// TIA Portal project "Alojado_FillingTank_FactoryIO" (V16)

(* hardware
DEVICE "S7-1200 station_1"  S7-1200 Station
   slot 0: "Rack_0"  S7-1200 Rack  Rack  V1.0
   slot 1: "PLC_1"  CPU 1215C DC/DC/DC  6ES7 215-1AG40-0XB0  V4.4
*)

// ===== PLC "PLC_1"  CPU 1215C DC/DC/DC =====

VAR_GLOBAL   // PLC tag table "Default tag table"
   "Tag_5" AT %M0.0 : Bool;
   "Tag_8" AT %M0.1 : Bool;
   "Tag_9" AT %MD10 : DInt;
   "Tag_10" AT %MD14 : DInt;
   "Tag_11" AT %MD18 : DInt;
   "Tag_1" AT %M0.2 : Bool;
   "Tag_12" AT %M0.3 : Bool;
   "Tag_13" AT %MD22 : Time;
   "Tag_14" AT %MD26 : DInt;
   "Tag_15" AT %MD30 : DInt;
END_VAR

VAR_GLOBAL   // PLC tag table "Tag table from XML_3"
   "Fill PB" AT %I10.0 : Bool;
   "Discharge PB" AT %I10.1 : Bool;
   "FACTORY I/O (Running)" AT %I10.2 : Bool;
   "Fill valve" AT %Q0.0 : Bool;
   "Filling Light" AT %Q0.1 : Bool;
   "Discharge valve" AT %Q0.2 : Bool;
   "Discharging Light" AT %Q0.3 : Bool;
   "Timer" AT %QD30 : DInt;
END_VAR

// folder: System blocks/Program resources

DATA_BLOCK "IEC_Timer_0_DB"   // DB1
{ S7_Optimized_Access := 'TRUE' }
AUTHOR : Simatic
FAMILY : IEC
NAME : IEC_TMR
VERSION : 1.0
// stored: InstanceOfName IEC_TIMER
"IEC_TIMER"
BEGIN
END_DATA_BLOCK

DATA_BLOCK "IEC_Timer_0_DB_1"   // DB2
{ S7_Optimized_Access := 'TRUE' }
AUTHOR : Simatic
FAMILY : IEC
NAME : IEC_TMR
VERSION : 1.0
// stored: InstanceOfName IEC_TIMER
"IEC_TIMER"
BEGIN
END_DATA_BLOCK

// folder: (top level)

FUNCTION "MHJ-PLC-Lab-Function-S71200" : Void   // FC9000, SCL
{ S7_Optimized_Access := 'TRUE' }
VERSION : 0.1
   VAR_TEMP
      rdTimeReturn : Int;
      outputTime : DTL;
      SyncVal : Byte;
      forVal : Int;
      forVal_2 : Int;
      Value : Byte;
   END_VAR
   VAR CONSTANT
      CompVal : Byte := 16#34;
      Value_01 : Byte := 16#11;
      Value_01_DW : DWord := 16#A165_D992;
      Value_02_DW : DWord := 16#58BE_4401;
   END_VAR
BEGIN

   #Value:=PEEK(area := 16#82,
        dbNumber := 0,
        byteOffset := 511);
   #Value := #Value + 1;

   POKE(area := 16#82,
        dbNumber := 0,
        byteOffset := 511,
        value := #Value);

   POKE(area:=16#81,
        dbNumber:=0,
        byteOffset:=1016,
        value:=#Value_01_DW);
   POKE(area := 16#81,
        dbNumber := 0,
        byteOffset := 1020,
        value := #Value_02_DW);

   POKE(area := 16#81,
        dbNumber := 0,
        byteOffset := 511,
        value := B#16#00);

   FOR #forVal := 0 TO 120 DO
       FOR #forVal_2:=0 TO 10 DO
           #rdTimeReturn:=RD_SYS_T(#outputTime);
           #rdTimeReturn := WR_SYS_T(#outputTime);
           #rdTimeReturn := RD_SYS_T(#outputTime);
           #rdTimeReturn := WR_SYS_T(#outputTime);
       END_FOR;
       #SyncVal:= PEEK(area := 16#81,
                      dbNumber := 0,
                      byteOffset := 511);
       IF #SyncVal = #CompVal THEN
          GOTO M_1;
       END_IF;
   END_FOR;
   RETURN;

   M_1:
   POKE(area := 16#81,
        dbNumber := 0,
        byteOffset := 511,
        value := B#16#0);
END_FUNCTION

ORGANIZATION_BLOCK "Main"   // OB1, LAD, ProgramCycle
TITLE = "Main Program Sweep (Cycle)"
{ S7_Optimized_Access := 'TRUE' }
VERSION : 0.1
   VAR_INPUT
      Initial_Call : Bool;   // Initial call of this OB
      Remanence : Bool;   // =True, if remanent data are available
   END_VAR
BEGIN

REGION Network 1
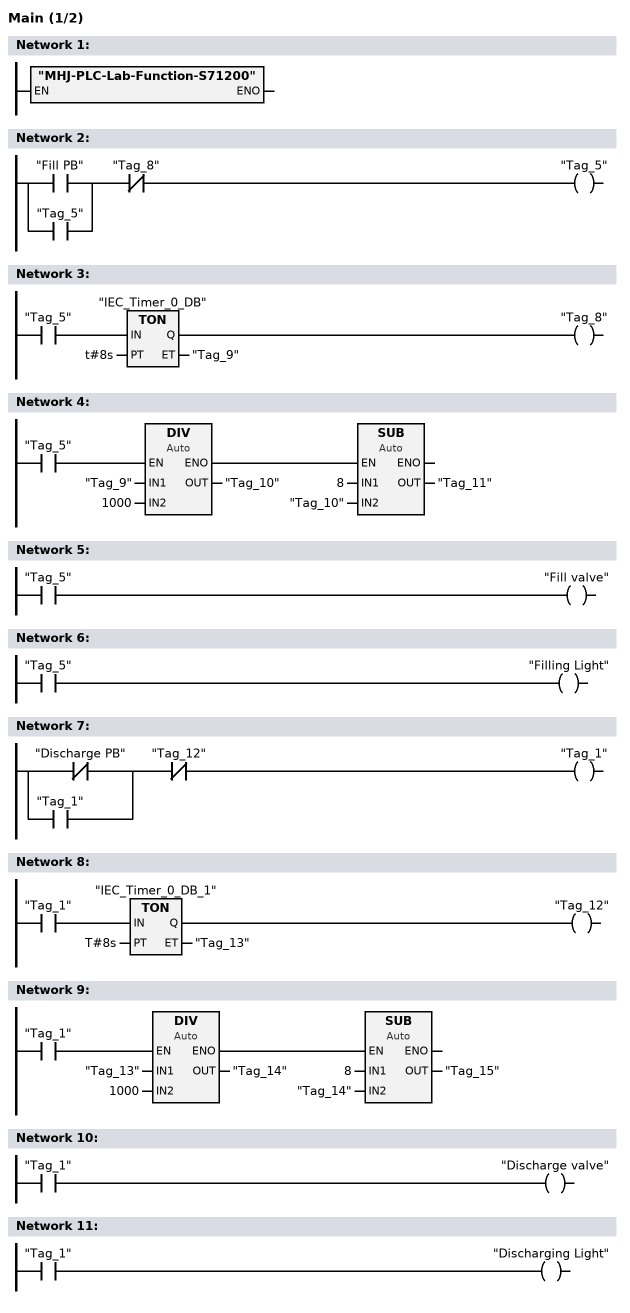
   RUNG wire#powerrail
      "MHJ-PLC-Lab-Function-S71200"()
   END_RUNG
   // the same network as SCL:
   "MHJ-PLC-Lab-Function-S71200"();
END_REGION

REGION Network 2
   RUNG wire#powerrail
      Contact( "Fill PB" )
      wire#w1
      I_Contact( "Tag_8" )
      Coil( "Tag_5" )
   END_RUNG
   RUNG wire#powerrail
      Contact( "Tag_5" )
   END_RUNG wire#w1
   // the same network as SCL:
   "Tag_5" := ("Fill PB" OR "Tag_5") AND NOT "Tag_8";
END_REGION

REGION Network 3
   "IEC_Timer_0_DB".TON(IN := "Tag_5", PT := t#8s, ET => "Tag_9");
   "Tag_8" := "IEC_Timer_0_DB".Q;
END_REGION

REGION Network 4
   RUNG wire#powerrail
      Contact( "Tag_5" )
      Div(in1 := "Tag_9", in2 := 1000, out => "Tag_10")
      Sub(in1 := 8, in2 := "Tag_10", out => "Tag_11")
   END_RUNG
   // the same network as SCL:
   IF "Tag_5" THEN
       "Tag_10" := "Tag_9" / 1000;
       "Tag_11" := 8 - "Tag_10";
   END_IF;
END_REGION

REGION Network 5
   RUNG wire#powerrail
      Contact( "Tag_5" )
      Coil( "Fill valve" )
   END_RUNG
   // the same network as SCL:
   "Fill valve" := "Tag_5";
END_REGION

REGION Network 6
   RUNG wire#powerrail
      Contact( "Tag_5" )
      Coil( "Filling Light" )
   END_RUNG
   // the same network as SCL:
   "Filling Light" := "Tag_5";
END_REGION

REGION Network 7
   RUNG wire#powerrail
      I_Contact( "Discharge PB" )
      wire#w1
      I_Contact( "Tag_12" )
      Coil( "Tag_1" )
   END_RUNG
   RUNG wire#powerrail
      Contact( "Tag_1" )
   END_RUNG wire#w1
   // the same network as SCL:
   "Tag_1" := (NOT "Discharge PB" OR "Tag_1") AND NOT "Tag_12";
END_REGION

REGION Network 8
   "IEC_Timer_0_DB_1".TON(IN := "Tag_1", PT := T#8s, ET => "Tag_13");
   "Tag_12" := "IEC_Timer_0_DB_1".Q;
END_REGION

REGION Network 9
   RUNG wire#powerrail
      Contact( "Tag_1" )
      Div(in1 := "Tag_13", in2 := 1000, out => "Tag_14")
      Sub(in1 := 8, in2 := "Tag_14", out => "Tag_15")
   END_RUNG
   // the same network as SCL:
   IF "Tag_1" THEN
       "Tag_14" := "Tag_13" / 1000;
       "Tag_15" := 8 - "Tag_14";
   END_IF;
END_REGION

REGION Network 10
   RUNG wire#powerrail
      Contact( "Tag_1" )
      Coil( "Discharge valve" )
   END_RUNG
   // the same network as SCL:
   "Discharge valve" := "Tag_1";
END_REGION

REGION Network 11
   RUNG wire#powerrail
      Contact( "Tag_1" )
      Coil( "Discharging Light" )
   END_RUNG
   // the same network as SCL:
   "Discharging Light" := "Tag_1";
END_REGION

REGION Network 12
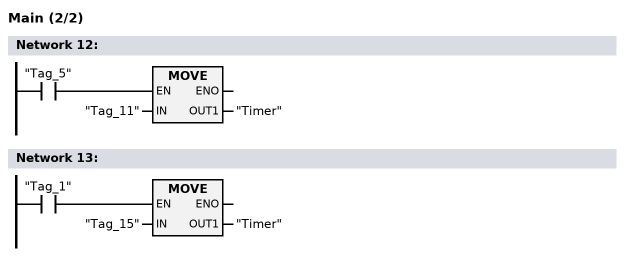
   RUNG wire#powerrail
      Contact( "Tag_5" )
      Move(in := "Tag_11", out1 => "Timer")
   END_RUNG
   // the same network as SCL:
   IF "Tag_5" THEN "Timer" := "Tag_11"; END_IF;
END_REGION

REGION Network 13
   RUNG wire#powerrail
      Contact( "Tag_1" )
      Move(in := "Tag_15", out1 => "Timer")
   END_RUNG
   // the same network as SCL:
   IF "Tag_1" THEN "Timer" := "Tag_15"; END_IF;
END_REGION
END_ORGANIZATION_BLOCK